FUNCTION_BLOCK FB_MotionLogger_TestDouble IMPLEMENTS I_MotionLogger
VAR
END_VAR

{warning 'Add method implementation '}
METHOD Clear
END_METHOD

METHOD ErrorCodeLookup : STRING
VAR_INPUT
	nErrorId	: UDINT;
END_VAR
END_METHOD

METHOD GetAllMessages :  STRING(1024)
END_METHOD

{warning 'Add method implementation '}
METHOD GetMessageCount : UINT
VAR_OUTPUT
	nCount	: UINT;
END_VAR
END_METHOD

{warning 'Add method implementation '}
METHOD Logger
VAR_INPUT
	Message	: STRING;
	Level	: E_MotionLogLevel := .E_MotionLogLevel.INFO;
	Source	: STRING := '';
END_VAR
END_METHOD

{warning 'Add property implementation'}
PROPERTY Name : STRING
GET
END_GET
END_PROPERTY

END_FUNCTION_BLOCK

(* stored: Version 1.1.0.1
   POU FB_MotionLogger_TestDouble: Id {8442344f-b7dd-4d6a-a684-1fd8fe76a797}, SpecialFunc None
   Method Clear: Id {700cd089-5255-48ab-b0ac-d9696853591e}
   Method ErrorCodeLookup: Id {57c70c9e-79a8-4868-91f2-6ad94f2941a5}
   Method GetAllMessages: Id {47b21366-5964-42c2-96e2-59304927e81d}
   Method GetMessageCount: Id {db2cfb9c-56db-4e54-ab8b-8b51ad930e34}
   Method Logger: Id {41b373f7-4e68-4a2f-bef2-7f808d9737a0}
   Property Name: Id {a1d48af6-c4e9-479f-8e5e-2c8e4f404352}
   Get Get: Id {7af4c83a-b130-4525-bb39-98ec1cdc3a66} *)
